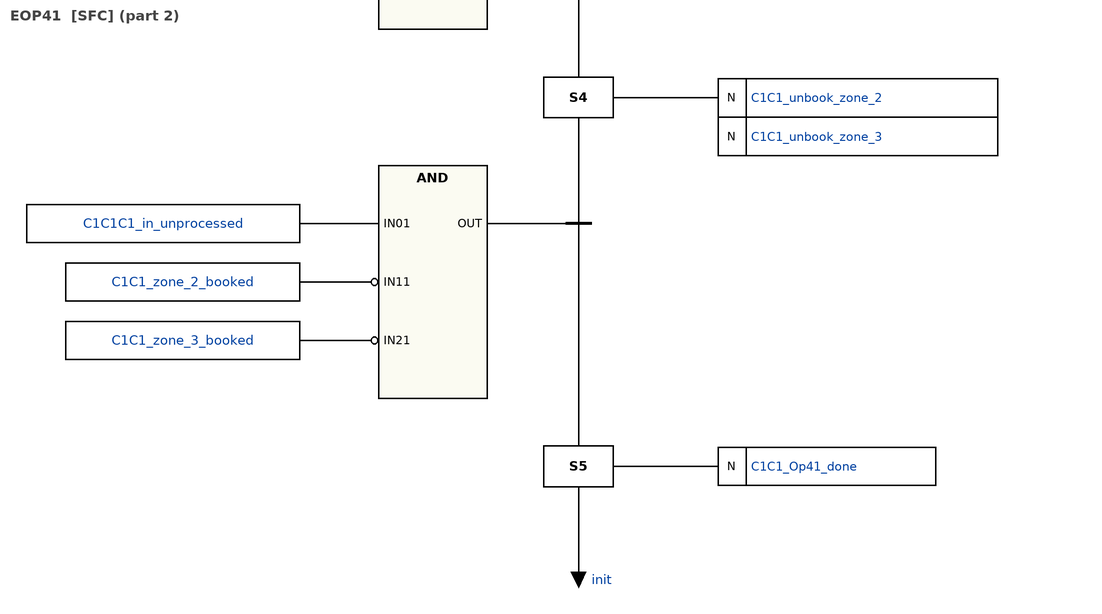
(* [picture p24: EOP41, SFC] *)
INITIAL_STEP init:
  COMPUTE_FUNCTION_BLOCKS(S);
END_STEP
TRANSITION FROM init TO S1
  := C1C1_Op41_exe_start;
END_TRANSITION
STEP S1:
END_STEP
TRANSITION FROM S1 TO S2
  := TRUE_VAR;
END_TRANSITION
STEP S2:
  C1C1_book_zone_2(N);
  C1C1_book_zone_3(N);
END_STEP
TRANSITION FROM S2 TO S3
  := _AND10_OUT;
END_TRANSITION
STEP S3:
  C1C1C1_goto_unprocessed(N);
END_STEP
TRANSITION FROM S3 TO S4
  := _AND16_OUT;
END_TRANSITION
STEP S4:
  C1C1_unbook_zone_2(N);
  C1C1_unbook_zone_3(N);
END_STEP
TRANSITION FROM S4 TO S5
  := _AND23_OUT;
END_TRANSITION
STEP S5:
  C1C1_Op41_done(N);
END_STEP
ACTION COMPUTE_FUNCTION_BLOCKS:  (* blocks drawn on the SFC sheet *)
  _AND10_OUT := C1C1_zone_2_booked AND C1C1_zone_3_booked;
  _AND16_OUT := C1C1C1_in_unprocessed AND C1C1_zone_2_booked AND C1C1_zone_3_booked;
  _AND23_OUT := C1C1C1_in_unprocessed AND NOT C1C1_zone_2_booked AND NOT C1C1_zone_3_booked;
END_ACTION
END_PROGRAM

PROGRAM EOP42
  VAR_EXTERNAL
    C1C1_Op42_exe_start : BOOL := false;
    TRUE_VAR : BOOL := true;
    C1C1C1_goto_processed : BOOL := false;
    C1C1C1_in_processed : BOOL := false;
    C1C1_Op42_done : BOOL := false;
  END_VAR

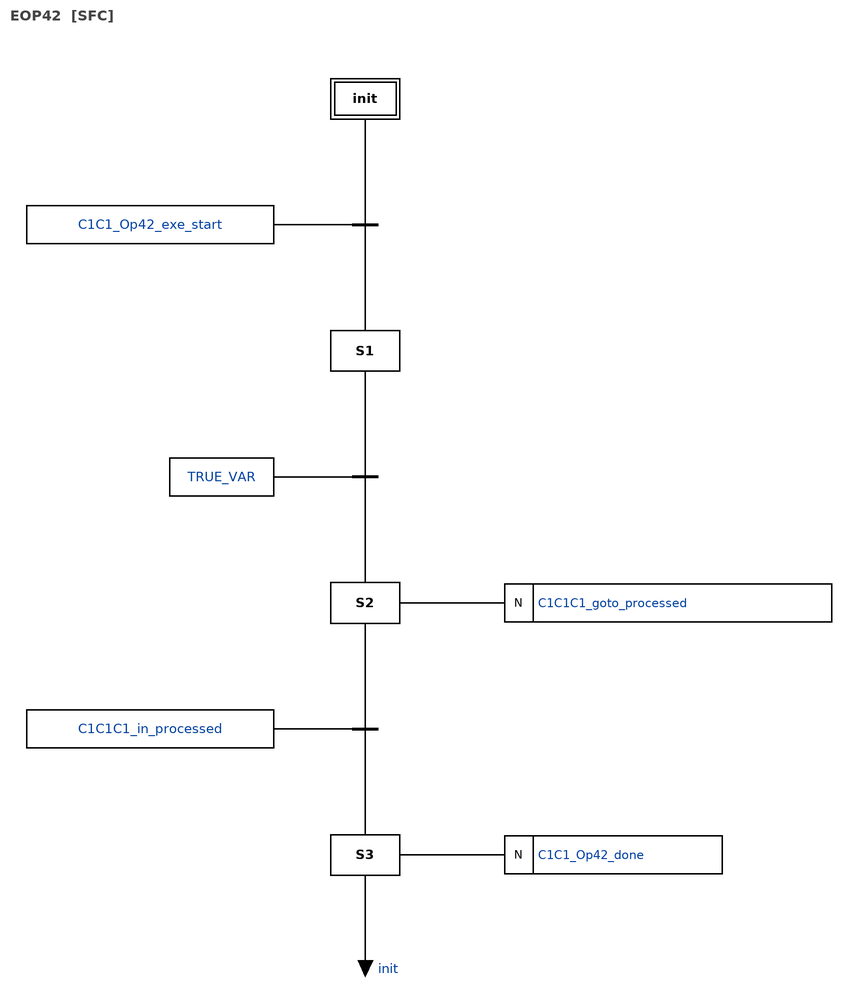
INITIAL_STEP init:
END_STEP
TRANSITION FROM init TO S1
  := C1C1_Op42_exe_start;
END_TRANSITION
STEP S1:
END_STEP
TRANSITION FROM S1 TO S2
  := TRUE_VAR;
END_TRANSITION
STEP S2:
  C1C1C1_goto_processed(N);
END_STEP
TRANSITION FROM S2 TO S3
  := C1C1C1_in_processed;
END_TRANSITION
STEP S3:
  C1C1_Op42_done(N);
END_STEP
END_PROGRAM

PROGRAM COP_C1C1_A
  VAR_EXTERNAL
    Start_COPs : BOOL := false;
    CC_A : BOOL := false;
    C1C1_Op40_exe_start : BOOL := false;
    C1C1_Op40_done : BOOL := false;
    C1C1_Op41_exe_start : BOOL := false;
    Op_34_end : BOOL := false;
    C1C1_Op41_done : BOOL := false;
    C1C1_Op42_exe_start : BOOL := false;
    C1C1_Op42_done : BOOL := false;
    COP_C1C1_A_done : BOOL := false;
    All_COP_Done_CC_A : BOOL := false;
  END_VAR
  VAR  (* added by the conversion: wires and edge detectors of the diagram *)
    _AND3_OUT : BOOL;
    _AND13_OUT : BOOL;
  END_VAR

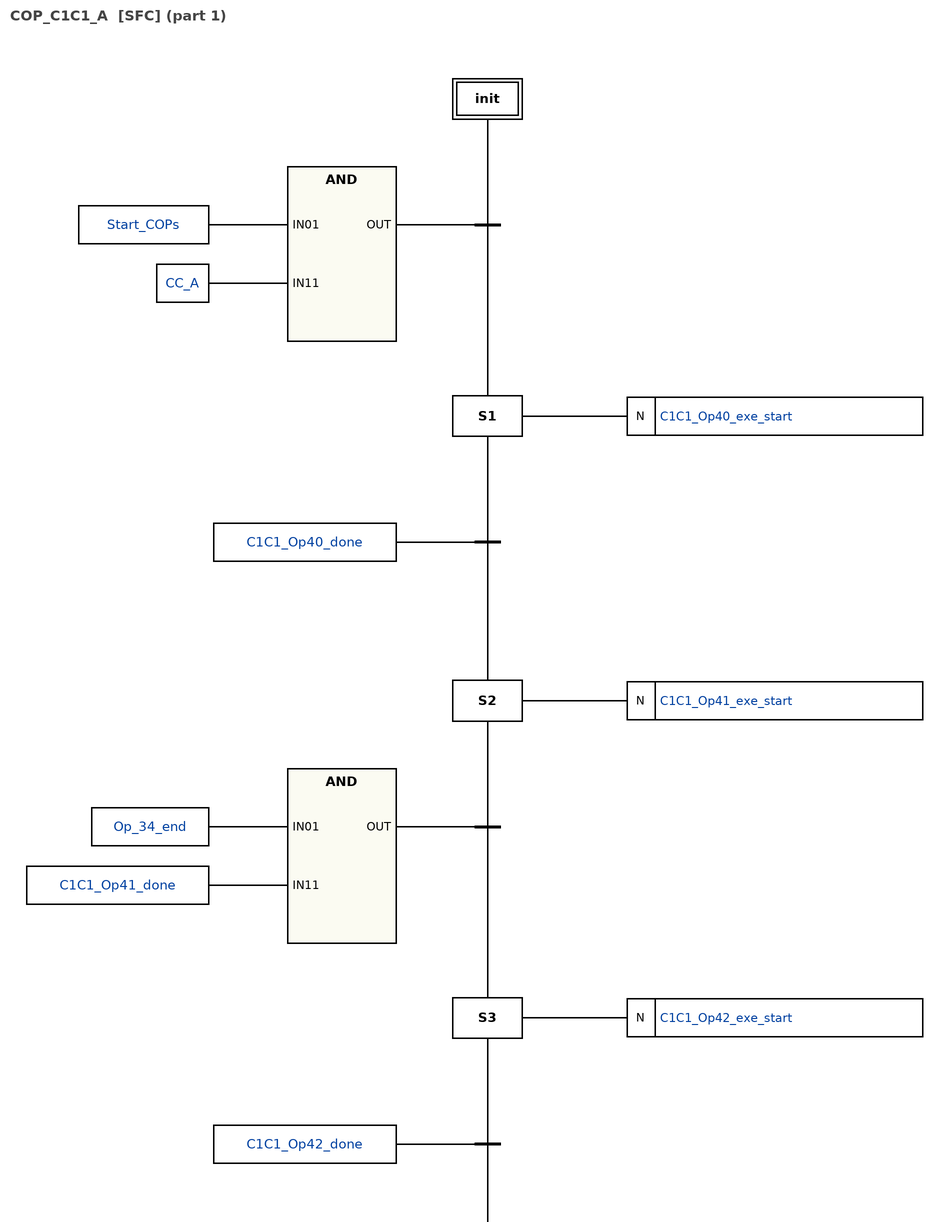
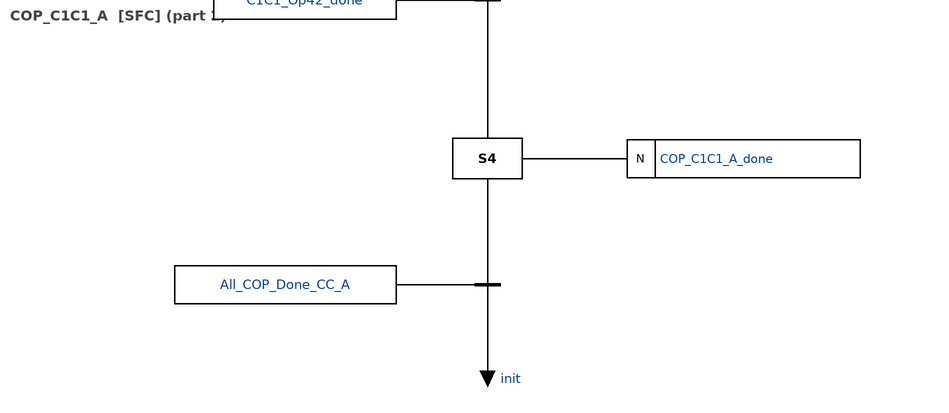
INITIAL_STEP init:
  COMPUTE_FUNCTION_BLOCKS(S);
END_STEP
TRANSITION FROM init TO S1
  := _AND3_OUT;
END_TRANSITION
STEP S1:
  C1C1_Op40_exe_start(N);
END_STEP
TRANSITION FROM S1 TO S2
  := C1C1_Op40_done;
END_TRANSITION
STEP S2:
  C1C1_Op41_exe_start(N);
END_STEP
TRANSITION FROM S2 TO S3
  := _AND13_OUT;
END_TRANSITION
STEP S3:
  C1C1_Op42_exe_start(N);
END_STEP
TRANSITION FROM S3 TO S4
  := C1C1_Op42_done;
END_TRANSITION
STEP S4:
  COP_C1C1_A_done(N);
END_STEP
TRANSITION FROM S4 TO init
  := All_COP_Done_CC_A;
END_TRANSITION
ACTION COMPUTE_FUNCTION_BLOCKS:  (* blocks drawn on the SFC sheet *)
  _AND3_OUT := Start_COPs AND CC_A;
  _AND13_OUT := Op_34_end AND C1C1_Op41_done;
END_ACTION
END_PROGRAM

PROGRAM COP_C1C1_B
  VAR_EXTERNAL
    Start_COPs : BOOL := false;
    CC_B : BOOL := false;
    C1C1_Op40_exe_start : BOOL := false;
    C1C1_Op40_done : BOOL := false;
    C1C1_Op43_exe_start : BOOL := false;
    C1C1_Op43_done : BOOL := false;
    COP_C1C1_B_done : BOOL := false;
    All_COP_Done_CC_B : BOOL := false;
  END_VAR
  VAR  (* added by the conversion: wires and edge detectors of the diagram *)
    _AND3_OUT : BOOL;
  END_VAR

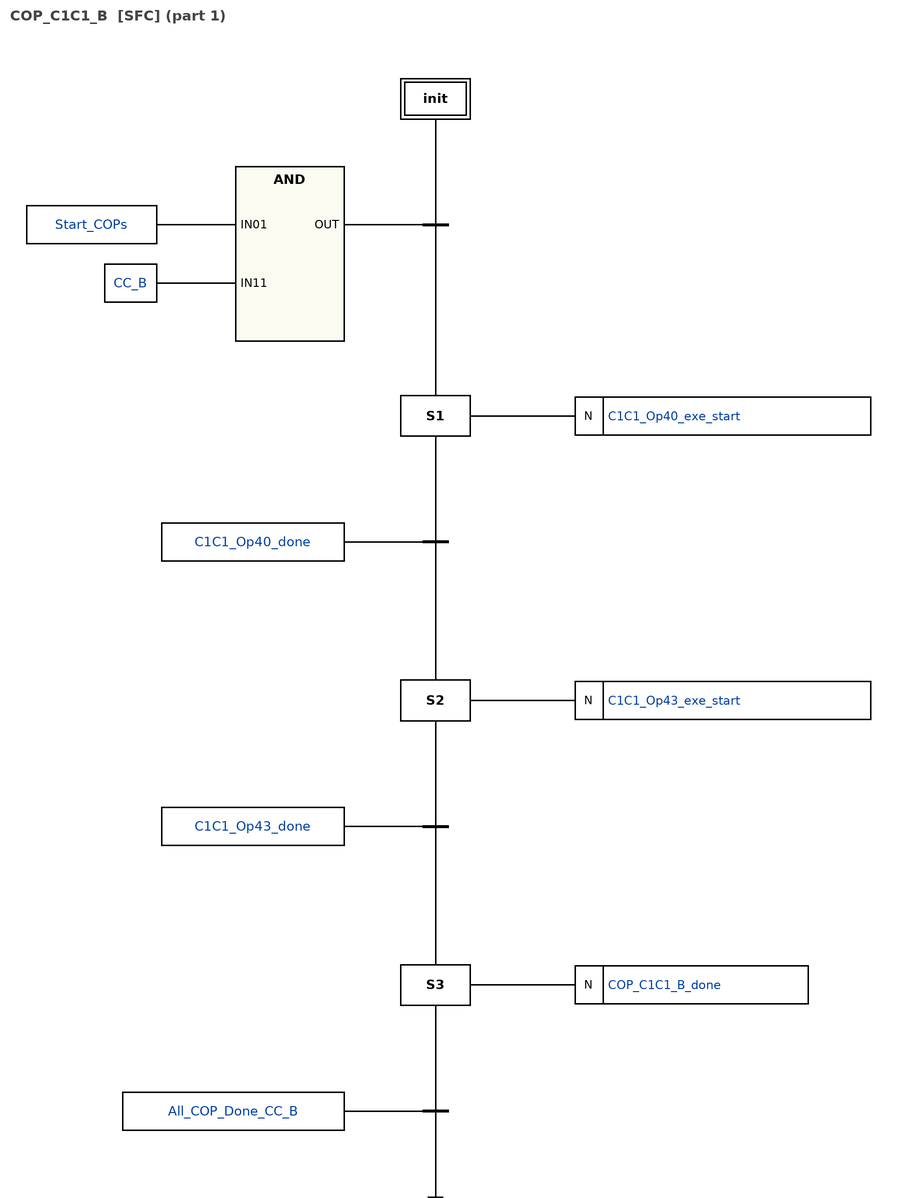
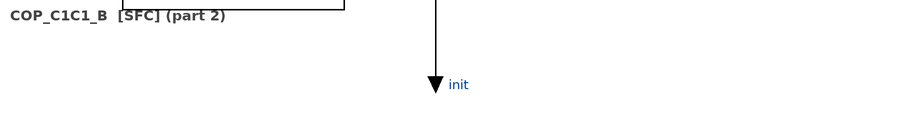
INITIAL_STEP init:
  COMPUTE_FUNCTION_BLOCKS(S);
END_STEP
TRANSITION FROM init TO S1
  := _AND3_OUT;
END_TRANSITION
STEP S1:
  C1C1_Op40_exe_start(N);
END_STEP
TRANSITION FROM S1 TO S2
  := C1C1_Op40_done;
END_TRANSITION
STEP S2:
  C1C1_Op43_exe_start(N);
END_STEP
TRANSITION FROM S2 TO S3
  := C1C1_Op43_done;
END_TRANSITION
STEP S3:
  COP_C1C1_B_done(N);
END_STEP
TRANSITION FROM S3 TO init
  := All_COP_Done_CC_B;
END_TRANSITION
ACTION COMPUTE_FUNCTION_BLOCKS:  (* blocks drawn on the SFC sheet *)
  _AND3_OUT := Start_COPs AND CC_B;
END_ACTION
END_PROGRAM

PROGRAM COP_C1C2_A
  VAR_EXTERNAL
    Start_COPs : BOOL := false;
    CC_A : BOOL := false;
    Op_10_start : BOOL := false;
    Op_10_end : BOOL := false;
    Op_11_start : BOOL := false;
    C1R1_Op21_done : BOOL := false;
    Op_11_end : BOOL := false;
    Op_12_start : BOOL := false;
    Op_12_end : BOOL := false;
    COP_C1C2_A_done : BOOL := false;
    All_COP_Done_CC_A : BOOL := false;
  END_VAR
  VAR  (* added by the conversion: wires and edge detectors of the diagram *)
    _AND3_OUT : BOOL;
    _AND13_OUT : BOOL;
  END_VAR

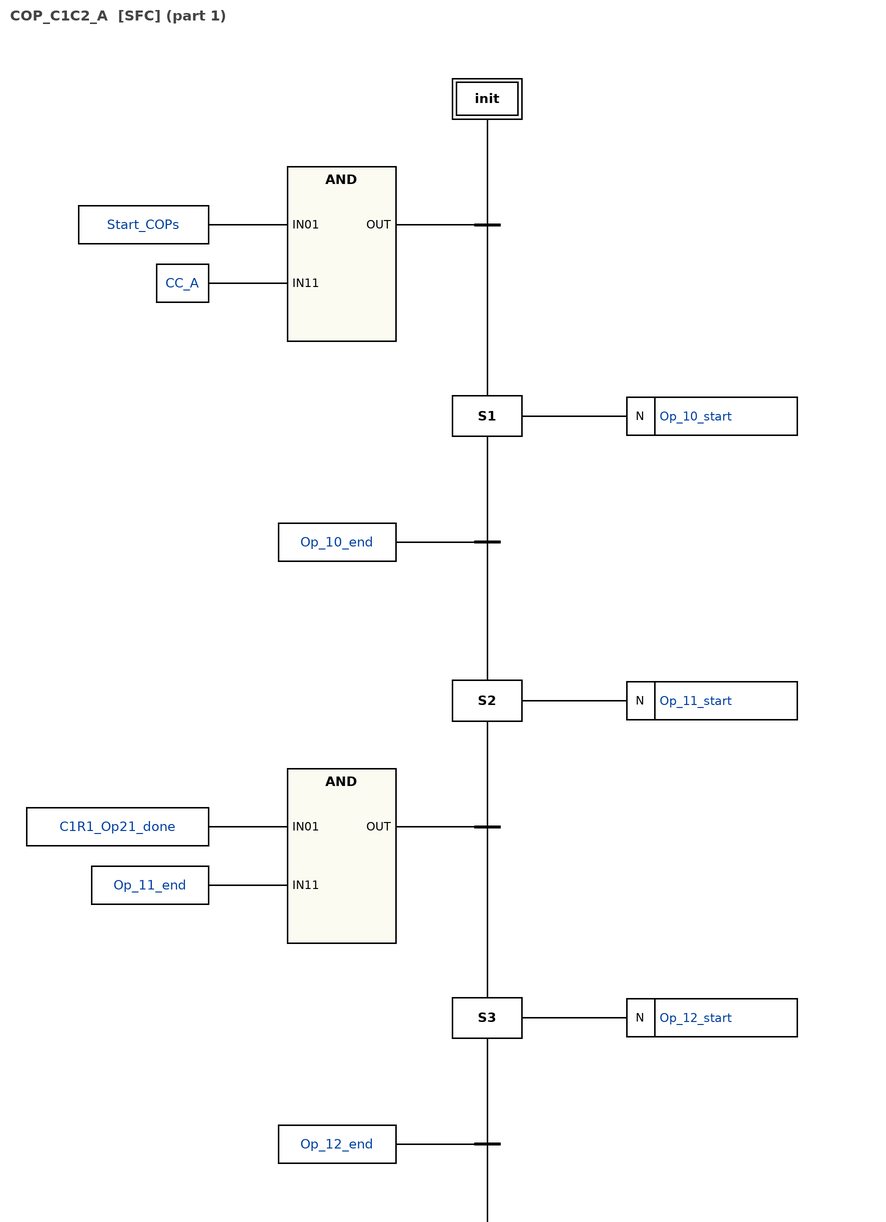
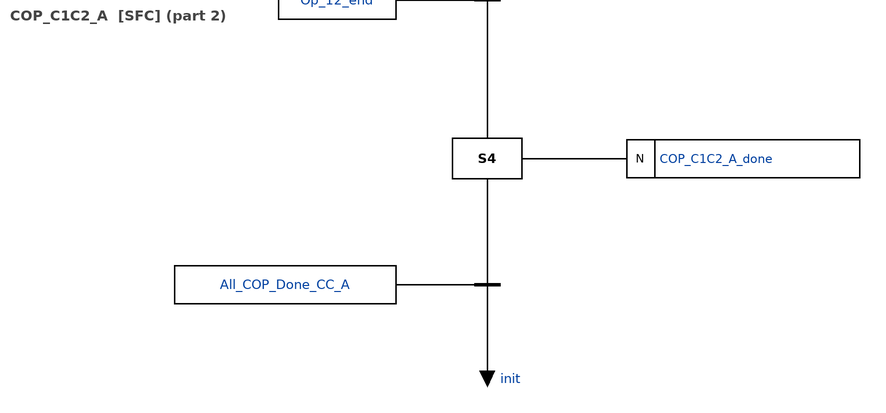
INITIAL_STEP init:
  COMPUTE_FUNCTION_BLOCKS(S);
END_STEP
TRANSITION FROM init TO S1
  := _AND3_OUT;
END_TRANSITION
STEP S1:
  Op_10_start(N);
END_STEP
TRANSITION FROM S1 TO S2
  := Op_10_end;
END_TRANSITION
STEP S2:
  Op_11_start(N);
END_STEP
TRANSITION FROM S2 TO S3
  := _AND13_OUT;
END_TRANSITION
STEP S3:
  Op_12_start(N);
END_STEP
TRANSITION FROM S3 TO S4
  := Op_12_end;
END_TRANSITION
STEP S4:
  COP_C1C2_A_done(N);
END_STEP
TRANSITION FROM S4 TO init
  := All_COP_Done_CC_A;
END_TRANSITION
ACTION COMPUTE_FUNCTION_BLOCKS:  (* blocks drawn on the SFC sheet *)
  _AND3_OUT := Start_COPs AND CC_A;
  _AND13_OUT := C1R1_Op21_done AND Op_11_end;
END_ACTION
END_PROGRAM

PROGRAM COP_C1C2_B
  VAR_EXTERNAL
    Start_COPs : BOOL := false;
    CC_B : BOOL := false;
    Op_10_start : BOOL := false;
    Op_10_end : BOOL := false;
    COP_C1C2_B_done : BOOL := false;
    All_COP_Done_CC_B : BOOL := false;
  END_VAR
  VAR  (* added by the conversion: wires and edge detectors of the diagram *)
    _AND3_OUT : BOOL;
  END_VAR

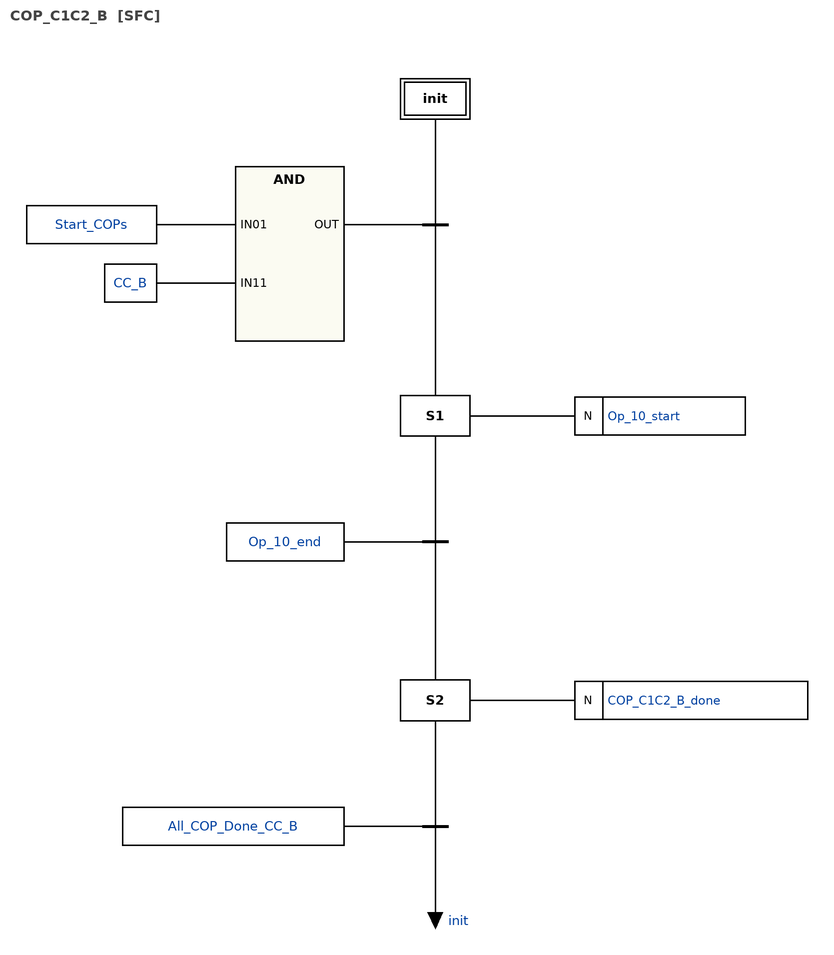
INITIAL_STEP init:
  COMPUTE_FUNCTION_BLOCKS(S);
END_STEP
TRANSITION FROM init TO S1
  := _AND3_OUT;
END_TRANSITION
STEP S1:
  Op_10_start(N);
END_STEP
TRANSITION FROM S1 TO S2
  := Op_10_end;
END_TRANSITION
STEP S2:
  COP_C1C2_B_done(N);
END_STEP
TRANSITION FROM S2 TO init
  := All_COP_Done_CC_B;
END_TRANSITION
ACTION COMPUTE_FUNCTION_BLOCKS:  (* blocks drawn on the SFC sheet *)
  _AND3_OUT := Start_COPs AND CC_B;
END_ACTION
END_PROGRAM

PROGRAM COP_C1F1_A
  VAR_EXTERNAL
    Start_COPs : BOOL := false;
    CC_A : BOOL := false;
    Op_30_start : BOOL := false;
    Op_30_end : BOOL := false;
    Op_31_start : BOOL := false;
    C1R1_Op22_done : BOOL := false;
    Op_31_end : BOOL := false;
    Op_32_start : BOOL := false;
    C1R1_Op23_done : BOOL := false;
    Op_32_end : BOOL := false;
    Op_33_start : BOOL := false;
    C1R1_Op24_done : BOOL := false;
    Op_33_end : BOOL := false;
    COP_C1F1_A_done : BOOL := false;
    All_COP_Done_CC_A : BOOL := false;
  END_VAR
  VAR  (* added by the conversion: wires and edge detectors of the diagram *)
    _AND3_OUT : BOOL;
    _AND13_OUT : BOOL;
    _AND19_OUT : BOOL;
    _AND25_OUT : BOOL;
  END_VAR

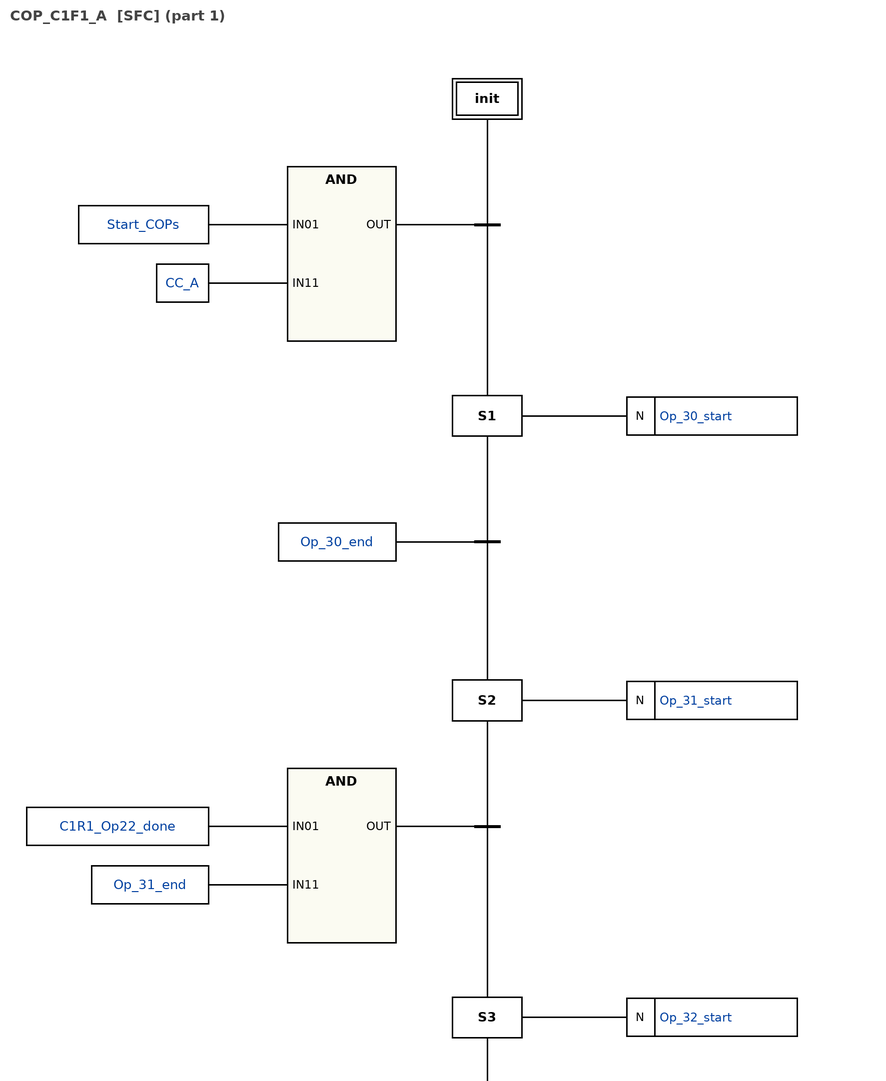
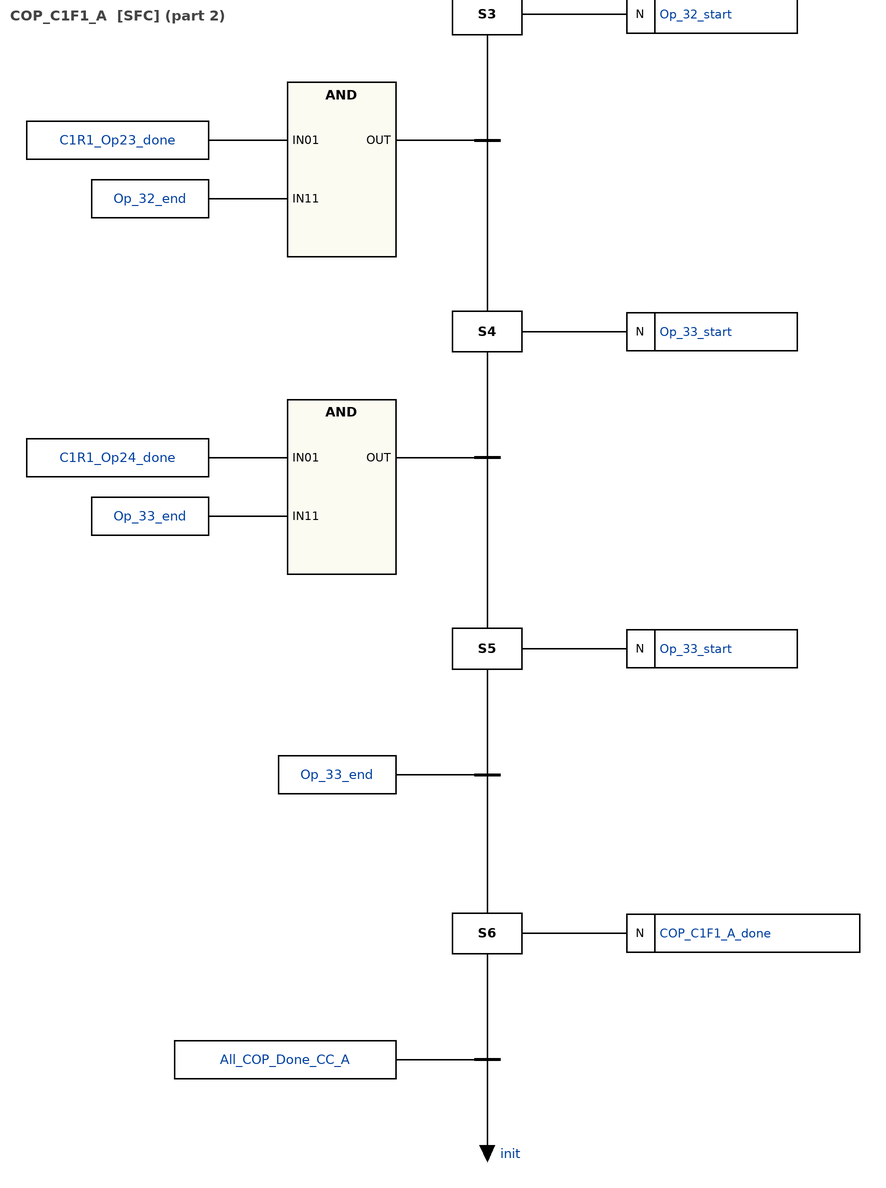
INITIAL_STEP init:
  COMPUTE_FUNCTION_BLOCKS(S);
END_STEP
TRANSITION FROM init TO S1
  := _AND3_OUT;
END_TRANSITION
STEP S1:
  Op_30_start(N);
END_STEP
TRANSITION FROM S1 TO S2
  := Op_30_end;
END_TRANSITION
STEP S2:
  Op_31_start(N);
END_STEP
TRANSITION FROM S2 TO S3
  := _AND13_OUT;
END_TRANSITION
STEP S3:
  Op_32_start(N);
END_STEP
TRANSITION FROM S3 TO S4
  := _AND19_OUT;
END_TRANSITION
STEP S4:
  Op_33_start(N);
END_STEP
TRANSITION FROM S4 TO S5
  := _AND25_OUT;
END_TRANSITION
STEP S5:
  Op_33_start(N);
END_STEP
TRANSITION FROM S5 TO S6
  := Op_33_end;
END_TRANSITION
STEP S6:
  COP_C1F1_A_done(N);
END_STEP
TRANSITION FROM S6 TO init
  := All_COP_Done_CC_A;
END_TRANSITION
ACTION COMPUTE_FUNCTION_BLOCKS:  (* blocks drawn on the SFC sheet *)
  _AND3_OUT := Start_COPs AND CC_A;
  _AND13_OUT := C1R1_Op22_done AND Op_31_end;
  _AND19_OUT := C1R1_Op23_done AND Op_32_end;
  _AND25_OUT := C1R1_Op24_done AND Op_33_end;
END_ACTION
END_PROGRAM

PROGRAM COP_C1F1_B
  VAR_EXTERNAL
    Start_COPs : BOOL := false;
    CC_B : BOOL := false;
    Op_30_start : BOOL := false;
    Op_30_end : BOOL := false;
    COP_C1F1_B_done : BOOL := false;
    All_COP_Done_CC_B : BOOL := false;
  END_VAR
  VAR  (* added by the conversion: wires and edge detectors of the diagram *)
    _AND3_OUT : BOOL;
  END_VAR

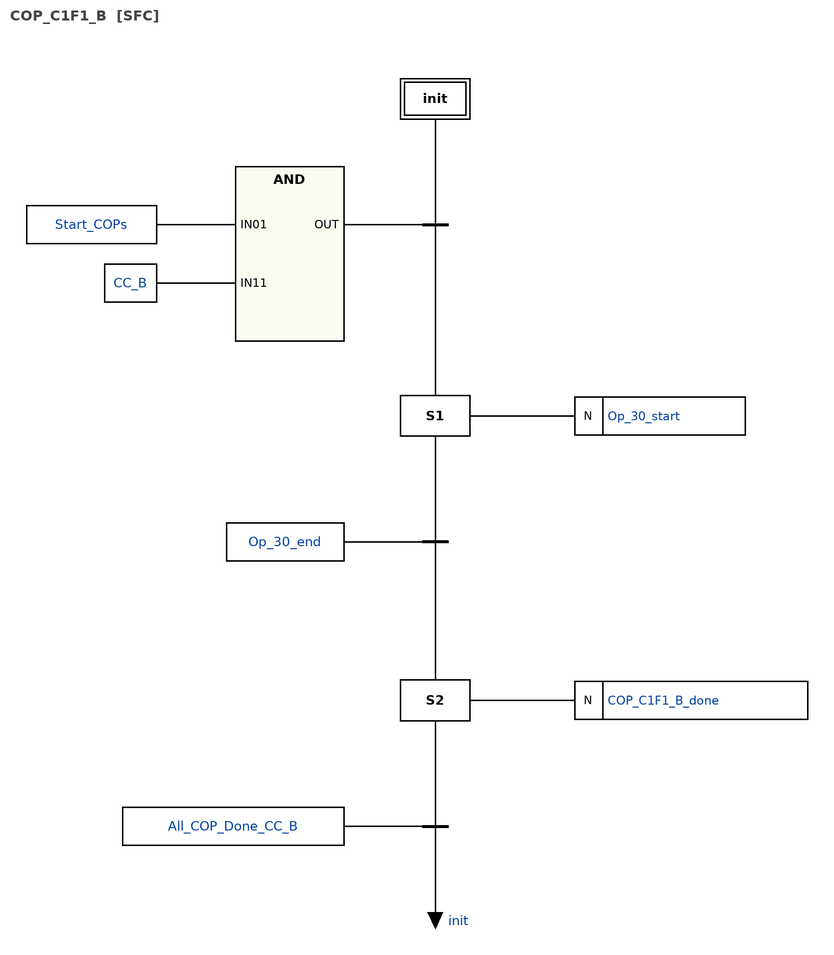
INITIAL_STEP init:
  COMPUTE_FUNCTION_BLOCKS(S);
END_STEP
TRANSITION FROM init TO S1
  := _AND3_OUT;
END_TRANSITION
STEP S1:
  Op_30_start(N);
END_STEP
TRANSITION FROM S1 TO S2
  := Op_30_end;
END_TRANSITION
STEP S2:
  COP_C1F1_B_done(N);
END_STEP
TRANSITION FROM S2 TO init
  := All_COP_Done_CC_B;
END_TRANSITION
ACTION COMPUTE_FUNCTION_BLOCKS:  (* blocks drawn on the SFC sheet *)
  _AND3_OUT := Start_COPs AND CC_B;
END_ACTION
END_PROGRAM

PROGRAM COP_C1R1_A
  VAR_EXTERNAL
    Start_COPs : BOOL := false;
    CC_A : BOOL := false;
    C1R1_Op20_exe_start : BOOL := false;
    Op_11_end : BOOL := false;
    C1R1_Op20_done : BOOL := false;
    C1R1_Op21_exe_start : BOOL := false;
    Op_31_end : BOOL := false;
    C1R1_Op21_done : BOOL := false;
    C1R1_Op22_exe_start : BOOL := false;
    Op_32_end : BOOL := false;
    C1R1_Op22_done : BOOL := false;
    C1R1_Op23_exe_start : BOOL := false;
    Op_33_end : BOOL := false;
    C1R1_Op23_done : BOOL := false;
    C1R1_Op24_exe_start : BOOL := false;
    C1R1_Op24_done : BOOL := false;
    COP_C1R1_A_done : BOOL := false;
    All_COP_Done_CC_A : BOOL := false;
  END_VAR
  VAR  (* added by the conversion: wires and edge detectors of the diagram *)
    _AND3_OUT : BOOL;
    _AND9_OUT : BOOL;
    _AND15_OUT : BOOL;
    _AND21_OUT : BOOL;
    _AND27_OUT : BOOL;
  END_VAR

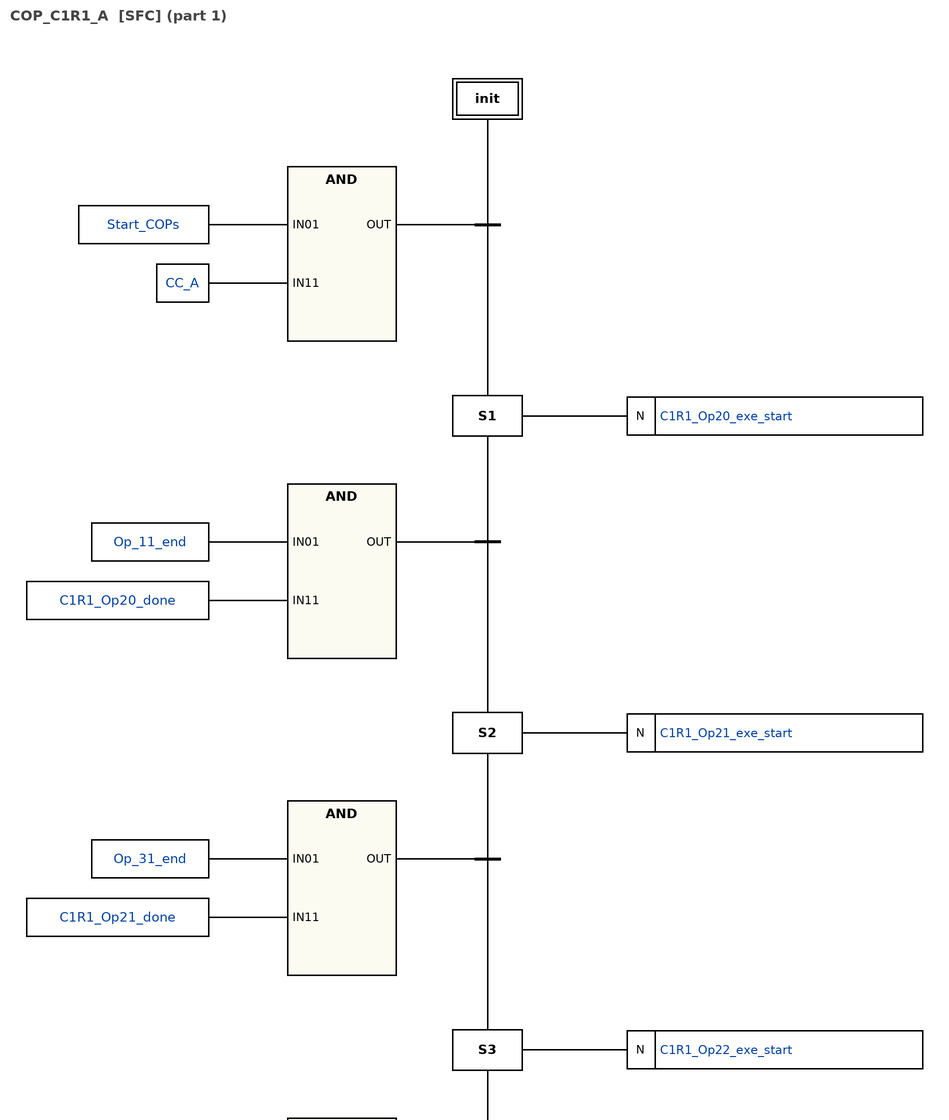
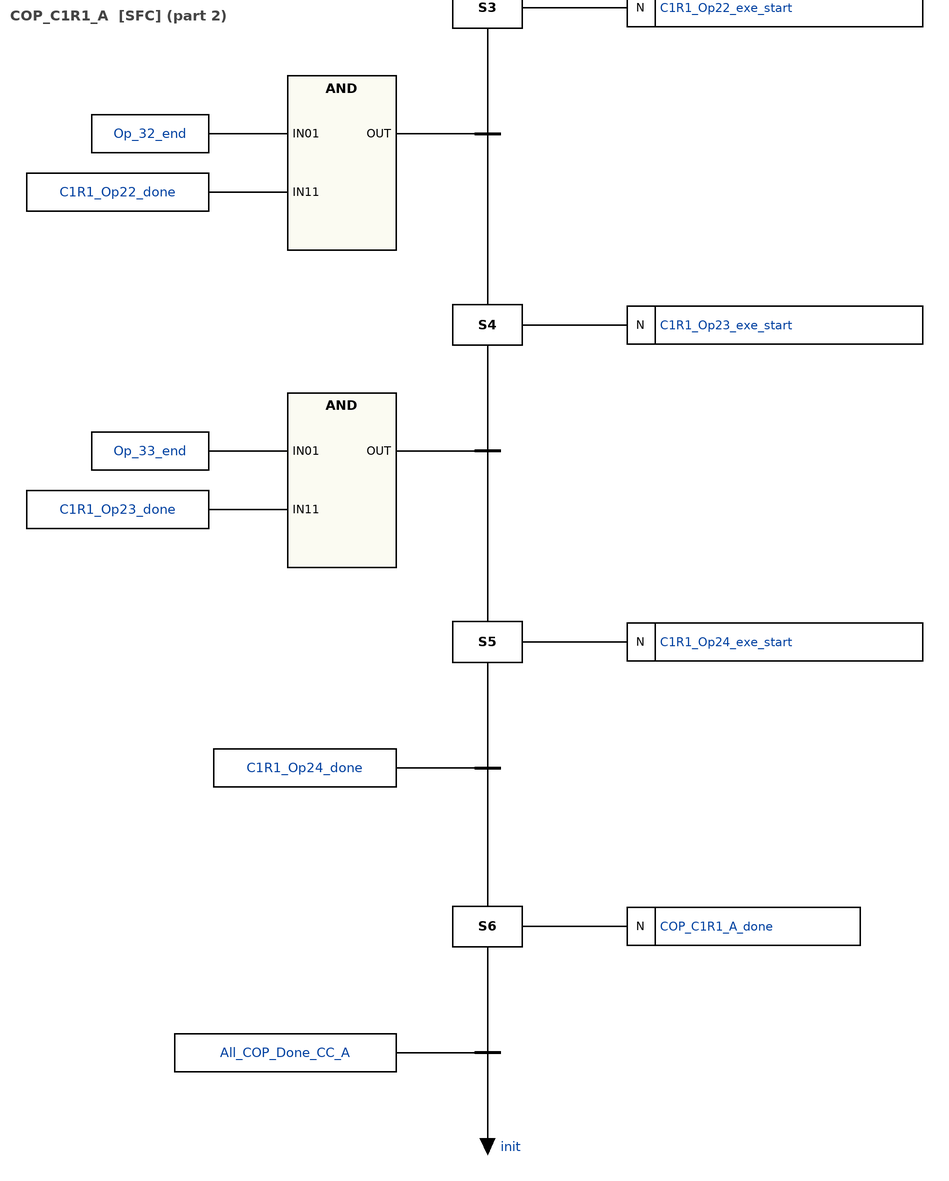
INITIAL_STEP init:
  COMPUTE_FUNCTION_BLOCKS(S);
END_STEP
TRANSITION FROM init TO S1
  := _AND3_OUT;
END_TRANSITION
STEP S1:
  C1R1_Op20_exe_start(N);
END_STEP
TRANSITION FROM S1 TO S2
  := _AND9_OUT;
END_TRANSITION
STEP S2:
  C1R1_Op21_exe_start(N);
END_STEP
TRANSITION FROM S2 TO S3
  := _AND15_OUT;
END_TRANSITION
STEP S3:
  C1R1_Op22_exe_start(N);
END_STEP
TRANSITION FROM S3 TO S4
  := _AND21_OUT;
END_TRANSITION
STEP S4:
  C1R1_Op23_exe_start(N);
END_STEP
TRANSITION FROM S4 TO S5
  := _AND27_OUT;
END_TRANSITION
STEP S5:
  C1R1_Op24_exe_start(N);
END_STEP
TRANSITION FROM S5 TO S6
  := C1R1_Op24_done;
END_TRANSITION
STEP S6:
  COP_C1R1_A_done(N);
END_STEP
TRANSITION FROM S6 TO init
  := All_COP_Done_CC_A;
END_TRANSITION
ACTION COMPUTE_FUNCTION_BLOCKS:  (* blocks drawn on the SFC sheet *)
  _AND3_OUT := Start_COPs AND CC_A;
  _AND9_OUT := Op_11_end AND C1R1_Op20_done;
  _AND15_OUT := Op_31_end AND C1R1_Op21_done;
  _AND21_OUT := Op_32_end AND C1R1_Op22_done;
  _AND27_OUT := Op_33_end AND C1R1_Op23_done;
END_ACTION
END_PROGRAM

PROGRAM FB_C1R1_External_Machine_comm_-_5_OP
  VAR_EXTERNAL
    C1R1_Op20_exe : BOOL := false;
    C1R1_Op20_IL : BOOL := false;
    C1R1_Op20_done : BOOL := false;
    C1R1_Op20_started : BOOL := false;
    C1R1_Op21_exe : BOOL := false;
    C1R1_Op21_IL : BOOL := false;
    C1R1_Op21_done : BOOL := false;
    C1R1_Op21_started : BOOL := false;
    C1R1_Op22_exe : BOOL := false;
    C1R1_Op22_IL : BOOL := false;
    C1R1_Op22_done : BOOL := false;
    C1R1_Op22_started : BOOL := false;
    C1R1_Op23_exe : BOOL := false;
    C1R1_Op23_IL : BOOL := false;
    C1R1_Op23_done : BOOL := false;
    C1R1_Op23_started : BOOL := false;
    C1R1_Op24_exe : BOOL := false;
    C1R1_Op24_IL : BOOL := false;
    C1R1_Op24_done : BOOL := false;
    C1R1_Op24_started : BOOL := false;
    C1R1_ext_lb_0 : BOOL := false;
    C1R1_ext_Ob_0 : BOOL := false;
    C1R1_ext_lb_1 : BOOL := false;
    C1R1_ext_Ob_1 : BOOL := false;
    C1R1_ext_lb_2 : BOOL := false;
    C1R1_ext_Ob_2 : BOOL := false;
    C1R1_ext_lb_3 : BOOL := false;
    C1R1_ext_Ob_3 : BOOL := false;
    C1R1_ext_lb_4 : BOOL := false;
    C1R1_ext_Ob_4 : BOOL := false;
    C1R1_ext_lb_5 : BOOL := false;
    C1R1_ext_Ob_5 : BOOL := false;
    C1R1_ext_lb_6 : BOOL := false;
    C1R1_ext_Ob_6 : BOOL := false;
    C1R1_ext_lb_7 : BOOL := false;
    C1R1_ext_Ob_7 : BOOL := false;
    C1R1_ext_machine_OK : BOOL := false;
    C1R1_IL_OK : BOOL := false;
  END_VAR
  VAR_EXTERNAL CONSTANT
    Constant_20 : INT := 20;
    Constant_21 : INT := 21;
    Constant_22 : INT := 22;
    Constant_23 : INT := 23;
    Constant_24 : INT := 24;
  END_VAR
  VAR
    FB_C1R1_External_Machine_comm_-_5_OP : External Machine comm - 5 OP;
  END_VAR

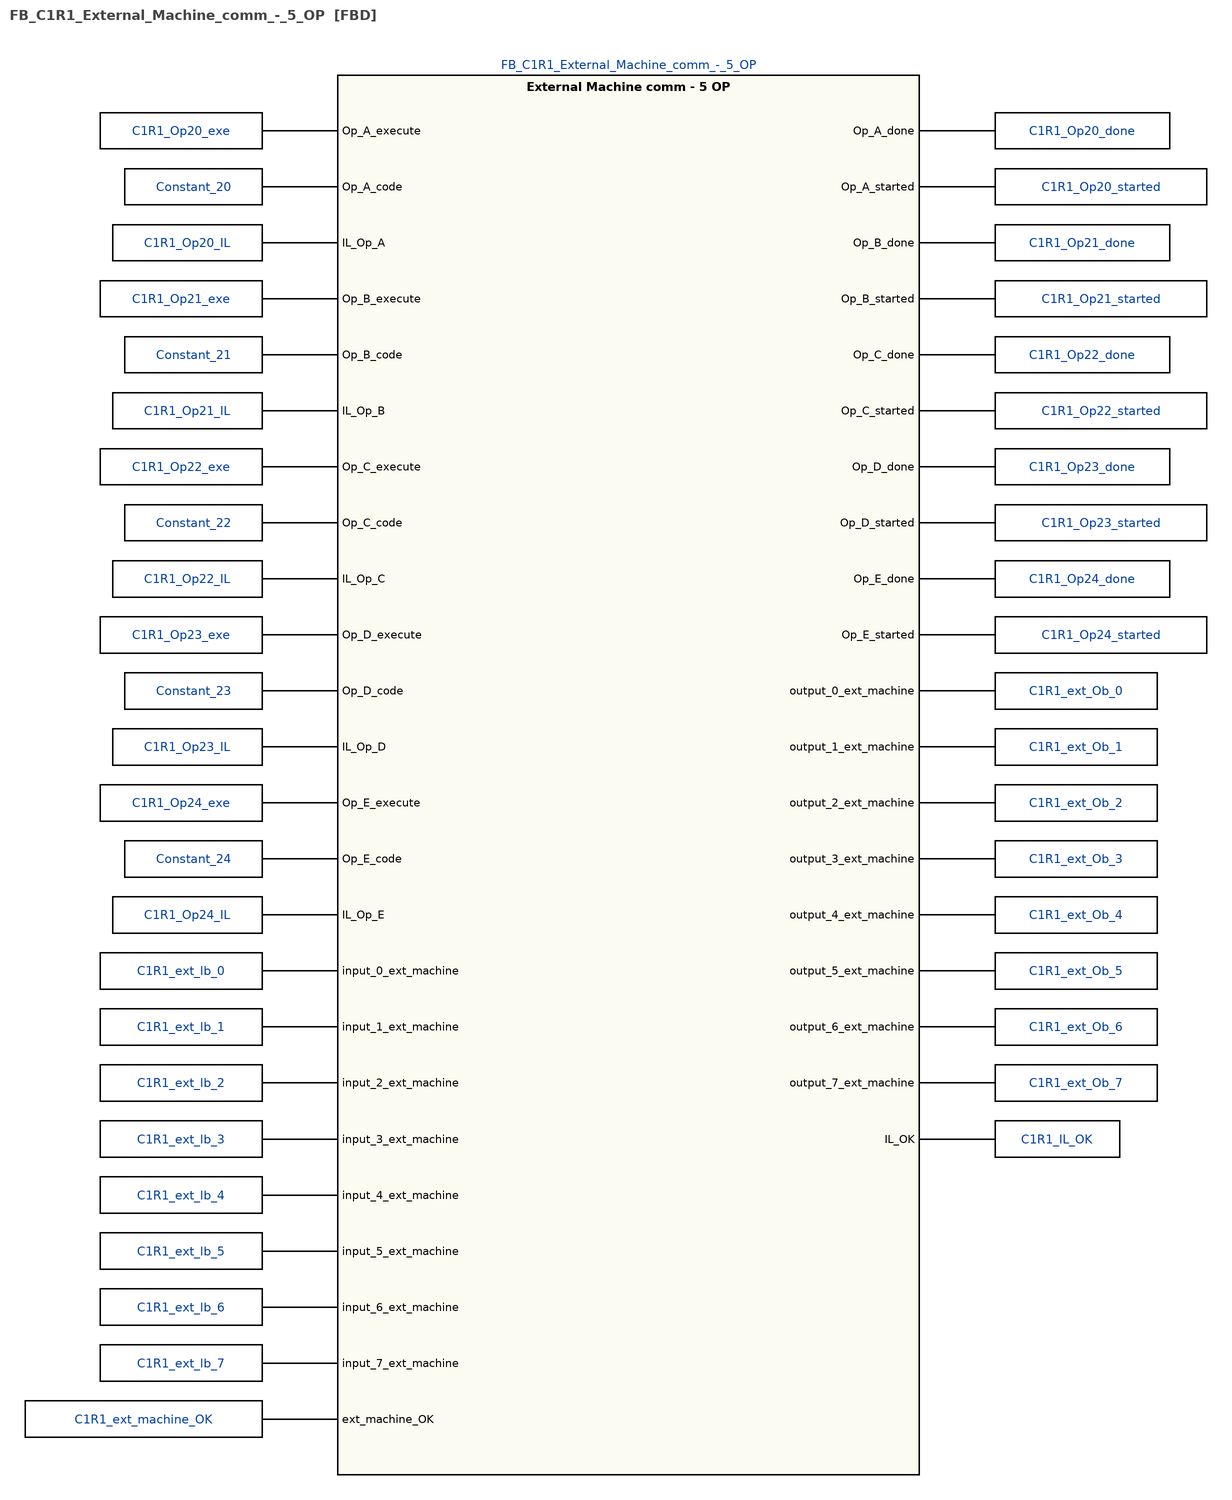
(* FBD diagram, written out as Structured Text *)
FB_C1R1_External_Machine_comm_-_5_OP(Op_A_execute := C1R1_Op20_exe, Op_A_code := Constant_20, IL_Op_A := C1R1_Op20_IL, Op_B_execute := C1R1_Op21_exe, Op_B_code := Constant_21, IL_Op_B := C1R1_Op21_IL, Op_C_execute := C1R1_Op22_exe, Op_C_code := Constant_22, IL_Op_C := C1R1_Op22_IL, Op_D_execute := C1R1_Op23_exe, Op_D_code := Constant_23, IL_Op_D := C1R1_Op23_IL, Op_E_execute := C1R1_Op24_exe, Op_E_code := Constant_24, IL_Op_E := C1R1_Op24_IL, input_0_ext_machine := C1R1_ext_lb_0, input_1_ext_machine := C1R1_ext_lb_1, input_2_ext_machine := C1R1_ext_lb_2, input_3_ext_machine := C1R1_ext_lb_3, input_4_ext_machine := C1R1_ext_lb_4, input_5_ext_machine := C1R1_ext_lb_5, input_6_ext_machine := C1R1_ext_lb_6, input_7_ext_machine := C1R1_ext_lb_7, ext_machine_OK := C1R1_ext_machine_OK);
C1R1_Op20_done := FB_C1R1_External_Machine_comm_-_5_OP.Op_A_done;
C1R1_Op20_started := FB_C1R1_External_Machine_comm_-_5_OP.Op_A_started;
C1R1_Op21_done := FB_C1R1_External_Machine_comm_-_5_OP.Op_B_done;
C1R1_Op21_started := FB_C1R1_External_Machine_comm_-_5_OP.Op_B_started;
C1R1_Op22_done := FB_C1R1_External_Machine_comm_-_5_OP.Op_C_done;
C1R1_Op22_started := FB_C1R1_External_Machine_comm_-_5_OP.Op_C_started;
C1R1_Op23_done := FB_C1R1_External_Machine_comm_-_5_OP.Op_D_done;
C1R1_Op23_started := FB_C1R1_External_Machine_comm_-_5_OP.Op_D_started;
C1R1_Op24_done := FB_C1R1_External_Machine_comm_-_5_OP.Op_E_done;
C1R1_Op24_started := FB_C1R1_External_Machine_comm_-_5_OP.Op_E_started;
C1R1_ext_Ob_0 := FB_C1R1_External_Machine_comm_-_5_OP.output_0_ext_machine;
C1R1_ext_Ob_1 := FB_C1R1_External_Machine_comm_-_5_OP.output_1_ext_machine;
C1R1_ext_Ob_2 := FB_C1R1_External_Machine_comm_-_5_OP.output_2_ext_machine;
C1R1_ext_Ob_3 := FB_C1R1_External_Machine_comm_-_5_OP.output_3_ext_machine;
C1R1_ext_Ob_4 := FB_C1R1_External_Machine_comm_-_5_OP.output_4_ext_machine;
C1R1_ext_Ob_5 := FB_C1R1_External_Machine_comm_-_5_OP.output_5_ext_machine;
C1R1_ext_Ob_6 := FB_C1R1_External_Machine_comm_-_5_OP.output_6_ext_machine;
C1R1_ext_Ob_7 := FB_C1R1_External_Machine_comm_-_5_OP.output_7_ext_machine;
C1R1_IL_OK := FB_C1R1_External_Machine_comm_-_5_OP.IL_OK;
END_PROGRAM

PROGRAM FB_C1C1_External_Machine_comm_-_4_OP
  VAR_EXTERNAL
    C1C1_Op40_exe : BOOL := false;
    C1C1_Op40_IL : BOOL := false;
    C1C1_Op40_done : BOOL := false;
    C1C1_Op40_started : BOOL := false;
    C1C1_Op41_exe : BOOL := false;
    C1C1_Op41_IL : BOOL := false;
    C1C1_Op41_done : BOOL := false;
    C1C1_Op41_started : BOOL := false;
    C1C1_Op42_exe : BOOL := false;
    C1C1_Op42_IL : BOOL := false;
    C1C1_Op42_done : BOOL := false;
    C1C1_Op42_started : BOOL := false;
    C1C1_Op43_exe : BOOL := false;
    C1C1_Op43_IL : BOOL := false;
    C1C1_Op43_done : BOOL := false;
    C1C1_Op43_started : BOOL := false;
    C1C1_ext_lb_0 : BOOL := false;
    C1C1_ext_Ob_0 : BOOL := false;
    C1C1_ext_lb_1 : BOOL := false;
    C1C1_ext_Ob_1 : BOOL := false;
    C1C1_ext_lb_2 : BOOL := false;
    C1C1_ext_Ob_2 : BOOL := false;
    C1C1_ext_lb_3 : BOOL := false;
    C1C1_ext_Ob_3 : BOOL := false;
    C1C1_ext_lb_4 : BOOL := false;
    C1C1_ext_Ob_4 : BOOL := false;
    C1C1_ext_lb_5 : BOOL := false;
    C1C1_ext_Ob_5 : BOOL := false;
    C1C1_ext_lb_6 : BOOL := false;
    C1C1_ext_Ob_6 : BOOL := false;
    C1C1_ext_lb_7 : BOOL := false;
    C1C1_ext_Ob_7 : BOOL := false;
    C1C1_ext_machine_OK : BOOL := false;
    C1C1_IL_OK : BOOL := false;
  END_VAR
  VAR_EXTERNAL CONSTANT
    Constant_40 : INT := 40;
    Constant_41 : INT := 41;
    Constant_42 : INT := 42;
    Constant_43 : INT := 43;
  END_VAR
  VAR
    FB_C1C1_External_Machine_comm_-_4_OP : External Machine comm - 4 OP;
  END_VAR

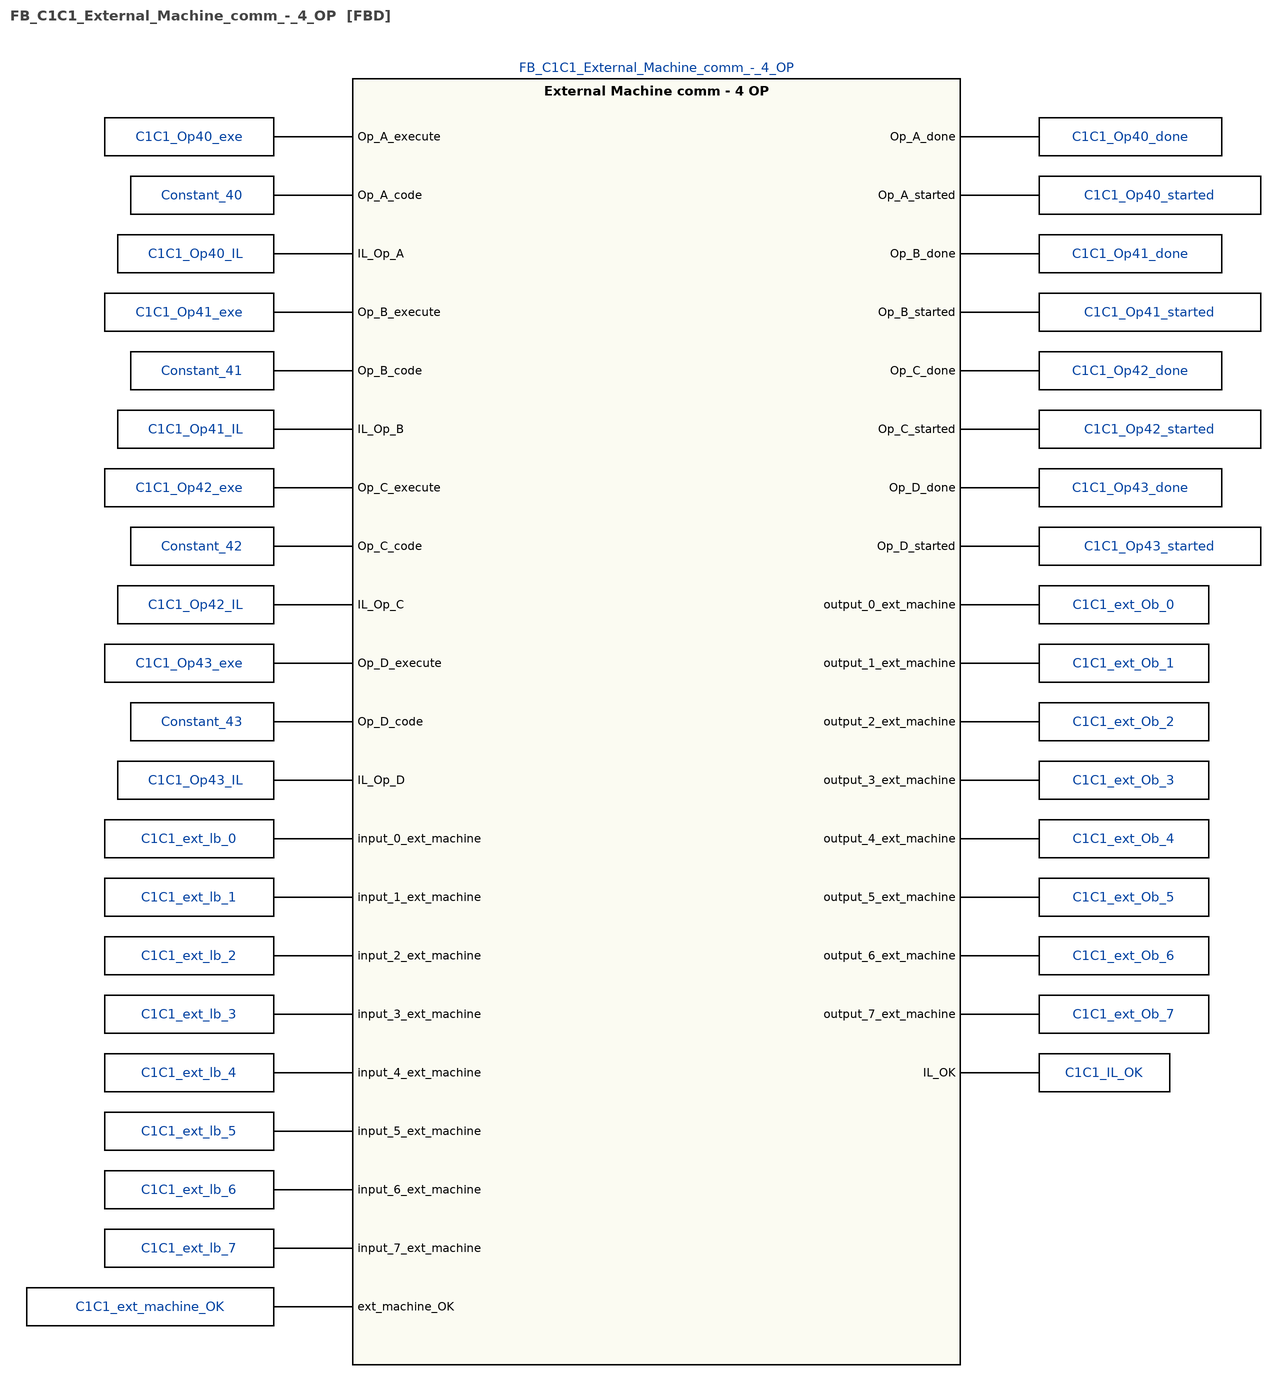
(* FBD diagram, written out as Structured Text *)
FB_C1C1_External_Machine_comm_-_4_OP(Op_A_execute := C1C1_Op40_exe, Op_A_code := Constant_40, IL_Op_A := C1C1_Op40_IL, Op_B_execute := C1C1_Op41_exe, Op_B_code := Constant_41, IL_Op_B := C1C1_Op41_IL, Op_C_execute := C1C1_Op42_exe, Op_C_code := Constant_42, IL_Op_C := C1C1_Op42_IL, Op_D_execute := C1C1_Op43_exe, Op_D_code := Constant_43, IL_Op_D := C1C1_Op43_IL, input_0_ext_machine := C1C1_ext_lb_0, input_1_ext_machine := C1C1_ext_lb_1, input_2_ext_machine := C1C1_ext_lb_2, input_3_ext_machine := C1C1_ext_lb_3, input_4_ext_machine := C1C1_ext_lb_4, input_5_ext_machine := C1C1_ext_lb_5, input_6_ext_machine := C1C1_ext_lb_6, input_7_ext_machine := C1C1_ext_lb_7, ext_machine_OK := C1C1_ext_machine_OK);
C1C1_Op40_done := FB_C1C1_External_Machine_comm_-_4_OP.Op_A_done;
C1C1_Op40_started := FB_C1C1_External_Machine_comm_-_4_OP.Op_A_started;
C1C1_Op41_done := FB_C1C1_External_Machine_comm_-_4_OP.Op_B_done;
C1C1_Op41_started := FB_C1C1_External_Machine_comm_-_4_OP.Op_B_started;
C1C1_Op42_done := FB_C1C1_External_Machine_comm_-_4_OP.Op_C_done;
C1C1_Op42_started := FB_C1C1_External_Machine_comm_-_4_OP.Op_C_started;
C1C1_Op43_done := FB_C1C1_External_Machine_comm_-_4_OP.Op_D_done;
C1C1_Op43_started := FB_C1C1_External_Machine_comm_-_4_OP.Op_D_started;
C1C1_ext_Ob_0 := FB_C1C1_External_Machine_comm_-_4_OP.output_0_ext_machine;
C1C1_ext_Ob_1 := FB_C1C1_External_Machine_comm_-_4_OP.output_1_ext_machine;
C1C1_ext_Ob_2 := FB_C1C1_External_Machine_comm_-_4_OP.output_2_ext_machine;
C1C1_ext_Ob_3 := FB_C1C1_External_Machine_comm_-_4_OP.output_3_ext_machine;
C1C1_ext_Ob_4 := FB_C1C1_External_Machine_comm_-_4_OP.output_4_ext_machine;
C1C1_ext_Ob_5 := FB_C1C1_External_Machine_comm_-_4_OP.output_5_ext_machine;
C1C1_ext_Ob_6 := FB_C1C1_External_Machine_comm_-_4_OP.output_6_ext_machine;
C1C1_ext_Ob_7 := FB_C1C1_External_Machine_comm_-_4_OP.output_7_ext_machine;
C1C1_IL_OK := FB_C1C1_External_Machine_comm_-_4_OP.IL_OK;
END_PROGRAM

PROGRAM FB_C1C2C1_Belt_Conveyor
  VAR_EXTERNAL
    C1C2C1_in_part_in_position : BOOL := false;
    C1C2C1_goto_part_in_position : BOOL := false;
    C1C2C1_IL_to_part_in_position : BOOL := false;
    C1C2C1_to_part_in_position_started : BOOL := false;
    C1C2C1_QS1 : BOOL := false;
    C1C2C1_in_position_empty : BOOL := false;
    C1C2C1_goto_position_empty : BOOL := false;
    C1C2C1_IL_to_position_empty : BOOL := false;
    C1C2C1_to_position_empty_started : BOOL := false;
    C1C2C1_QS2 : BOOL := false;
    Not_Connected : BOOL := false;
  END_VAR
  VAR
    FB_C1C2C1_Belt_Conveyor : Belt Conveyor;
  END_VAR

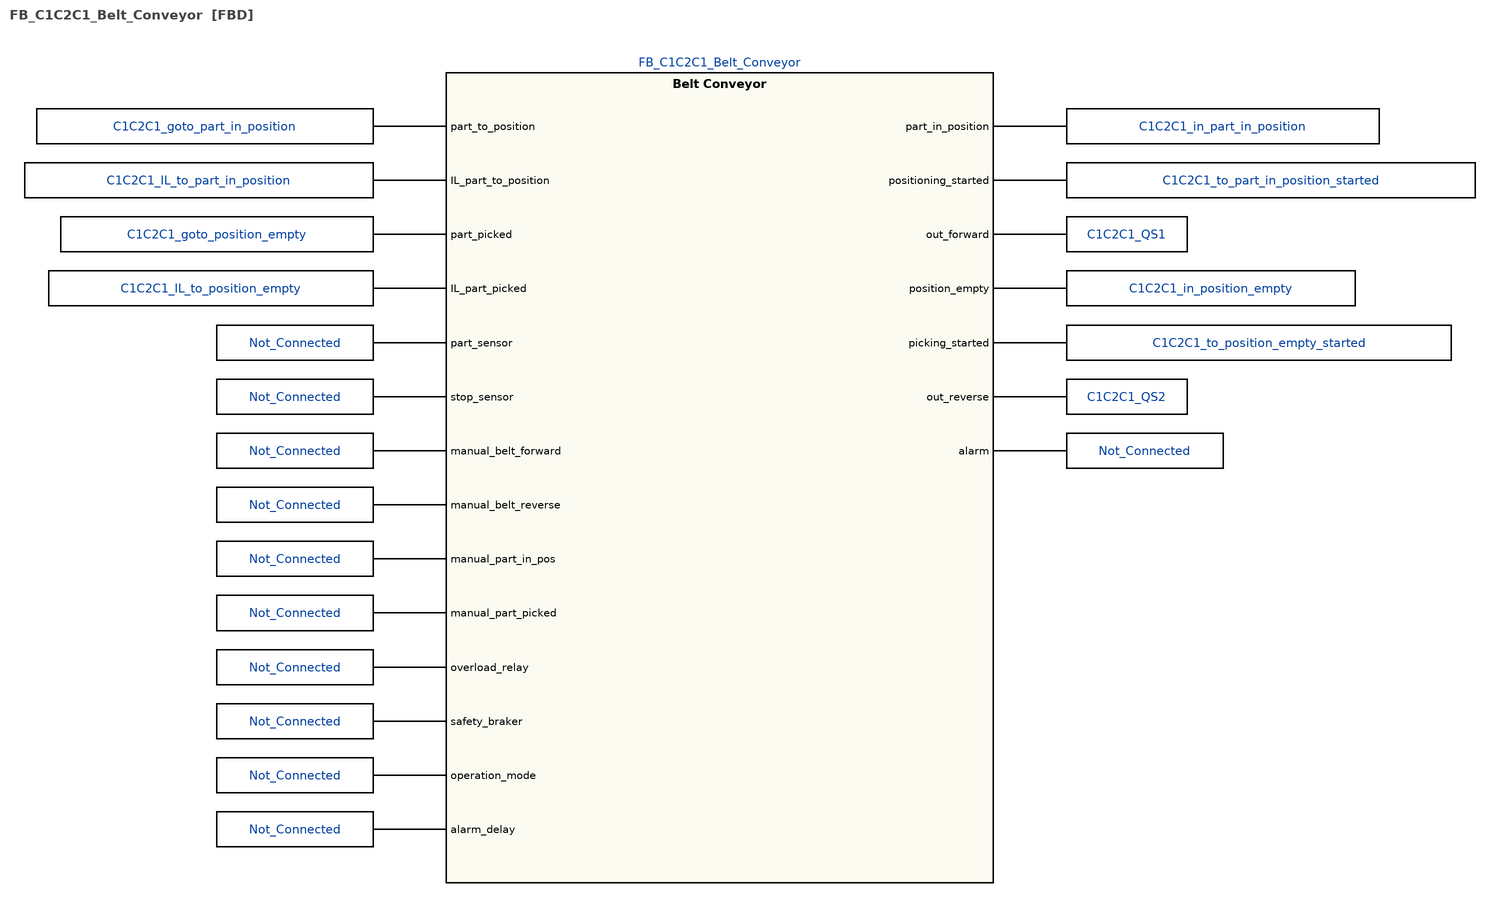
(* FBD diagram, written out as Structured Text *)
FB_C1C2C1_Belt_Conveyor(part_to_position := C1C2C1_goto_part_in_position, IL_part_to_position := C1C2C1_IL_to_part_in_position, part_picked := C1C2C1_goto_position_empty, IL_part_picked := C1C2C1_IL_to_position_empty, part_sensor := Not_Connected, stop_sensor := Not_Connected, manual_belt_forward := Not_Connected, manual_belt_reverse := Not_Connected, manual_part_in_pos := Not_Connected, manual_part_picked := Not_Connected, overload_relay := Not_Connected, safety_braker := Not_Connected, operation_mode := Not_Connected, alarm_delay := Not_Connected);
C1C2C1_in_part_in_position := FB_C1C2C1_Belt_Conveyor.part_in_position;
C1C2C1_to_part_in_position_started := FB_C1C2C1_Belt_Conveyor.positioning_started;
C1C2C1_QS1 := FB_C1C2C1_Belt_Conveyor.out_forward;
C1C2C1_in_position_empty := FB_C1C2C1_Belt_Conveyor.position_empty;
C1C2C1_to_position_empty_started := FB_C1C2C1_Belt_Conveyor.picking_started;
C1C2C1_QS2 := FB_C1C2C1_Belt_Conveyor.out_reverse;
Not_Connected := FB_C1C2C1_Belt_Conveyor.alarm;
END_PROGRAM

PROGRAM FB_C1F1C1_Two_Position_Movement
  VAR_EXTERNAL
    C1F1C1_in_home : BOOL := false;
    C1F1C1_goto_home : BOOL := false;
    C1F1C1_IL_to_home : BOOL := false;
    C1F1C1_to_home_started : BOOL := false;
    C1F1C1_QS1 : BOOL := false;
    C1F1C1_IS1 : BOOL := false;
    C1F1C1_in_work_pos : BOOL := false;
    C1F1C1_goto_work_pos : BOOL := false;
    C1F1C1_IL_to_work_pos : BOOL := false;
    C1F1C1_to_work_pos_started : BOOL := false;
    C1F1C1_QS2 : BOOL := false;
    C1F1C1_IS2 : BOOL := false;
    Not_Connected : BOOL := false;
  END_VAR
  VAR
    FB_C1F1C1_Two_Position_Movement : Two Position Movement;
  END_VAR

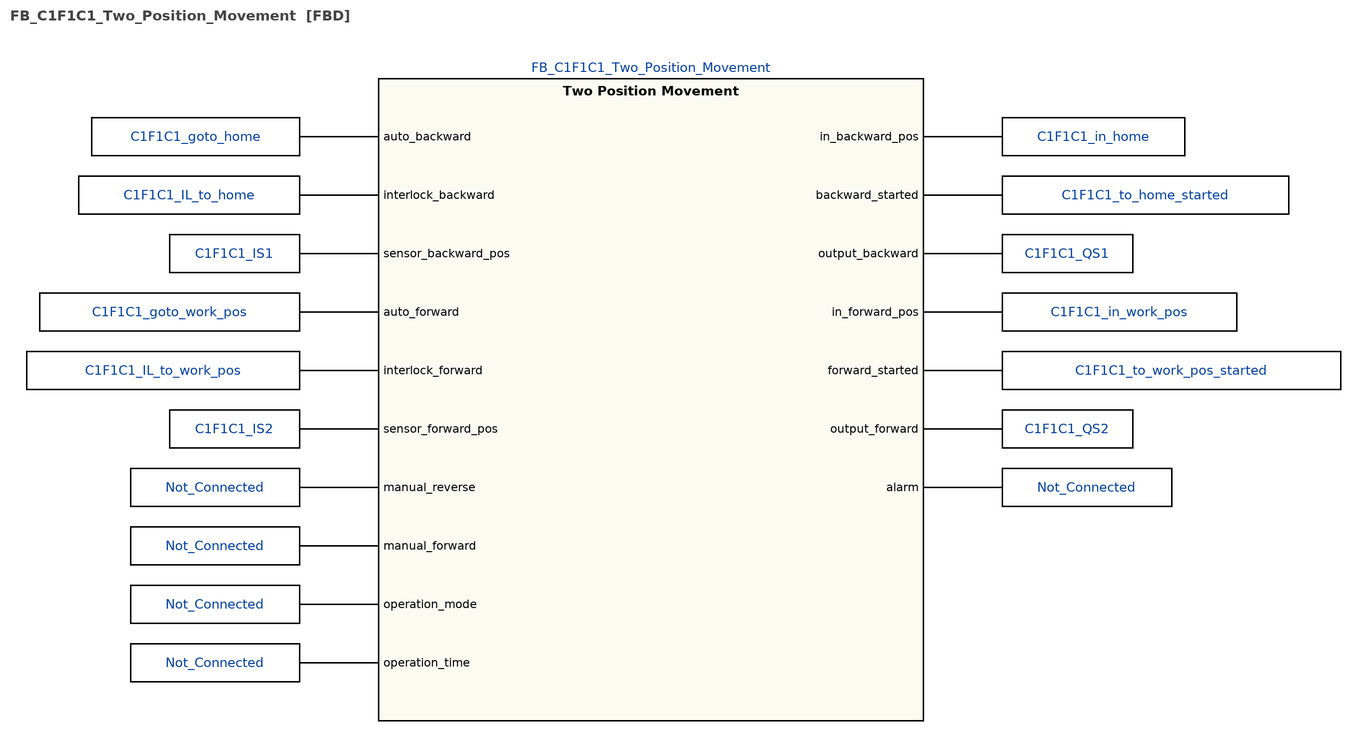
(* FBD diagram, written out as Structured Text *)
FB_C1F1C1_Two_Position_Movement(auto_backward := C1F1C1_goto_home, interlock_backward := C1F1C1_IL_to_home, sensor_backward_pos := C1F1C1_IS1, auto_forward := C1F1C1_goto_work_pos, interlock_forward := C1F1C1_IL_to_work_pos, sensor_forward_pos := C1F1C1_IS2, manual_reverse := Not_Connected, manual_forward := Not_Connected, operation_mode := Not_Connected, operation_time := Not_Connected);
C1F1C1_in_home := FB_C1F1C1_Two_Position_Movement.in_backward_pos;
C1F1C1_to_home_started := FB_C1F1C1_Two_Position_Movement.backward_started;
C1F1C1_QS1 := FB_C1F1C1_Two_Position_Movement.output_backward;
C1F1C1_in_work_pos := FB_C1F1C1_Two_Position_Movement.in_forward_pos;
C1F1C1_to_work_pos_started := FB_C1F1C1_Two_Position_Movement.forward_started;
C1F1C1_QS2 := FB_C1F1C1_Two_Position_Movement.output_forward;
Not_Connected := FB_C1F1C1_Two_Position_Movement.alarm;
END_PROGRAM

PROGRAM FB_C1F1C2_Two_Position_Movement
  VAR_EXTERNAL
    C1F1C2_in_locked : BOOL := false;
    C1F1C2_goto_locked : BOOL := false;
    C1F1C2_IL_to_locked : BOOL := false;
    C1F1C2_to_locked_started : BOOL := false;
    C1F1C2_QS1 : BOOL := false;
    C1F1C2_IS1 : BOOL := false;
    C1F1C2_in_unlocked : BOOL := false;
    C1F1C2_goto_unlocked : BOOL := false;
    C1F1C2_IL_to_unlocked : BOOL := false;
    C1F1C2_to_unlocked_started : BOOL := false;
    C1F1C2_QS2 : BOOL := false;
    C1F1C2_IS2 : BOOL := false;
    Not_Connected : BOOL := false;
  END_VAR
  VAR
    FB_C1F1C2_Two_Position_Movement : Two Position Movement;
  END_VAR

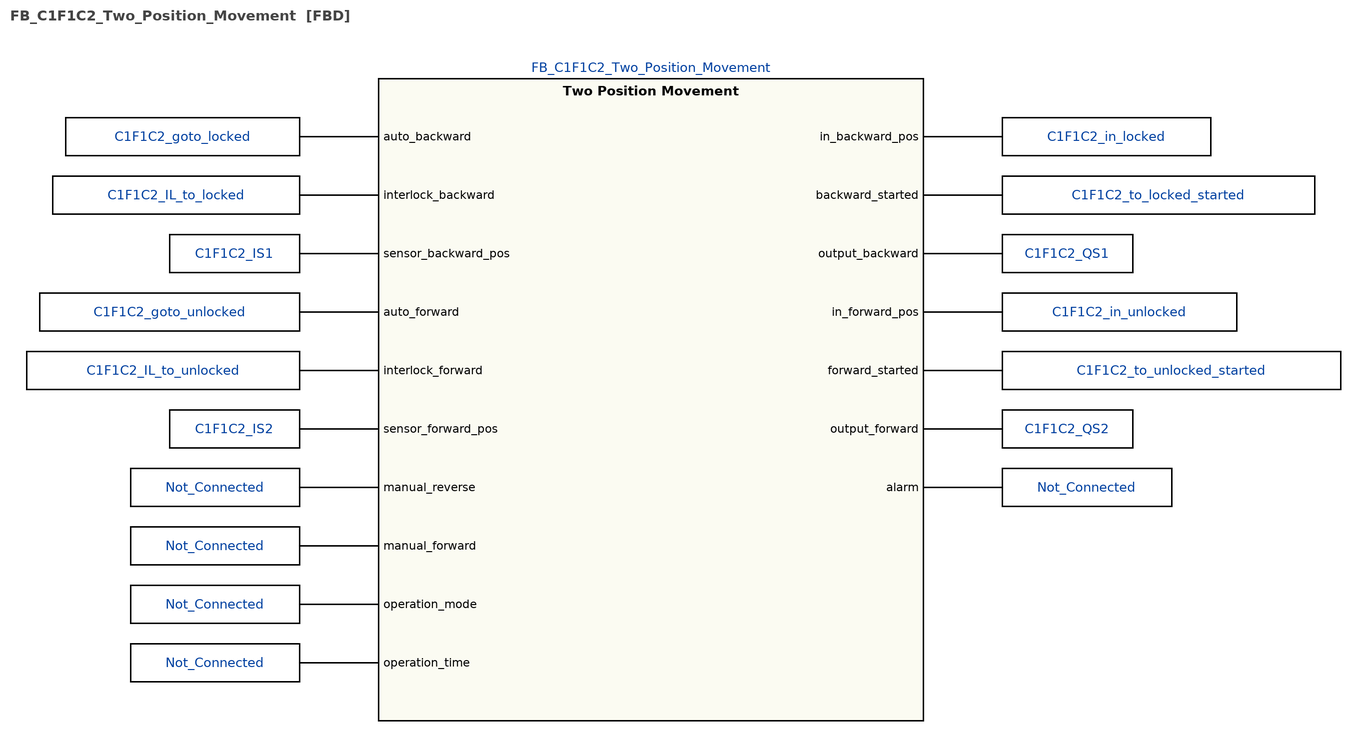
(* FBD diagram, written out as Structured Text *)
FB_C1F1C2_Two_Position_Movement(auto_backward := C1F1C2_goto_locked, interlock_backward := C1F1C2_IL_to_locked, sensor_backward_pos := C1F1C2_IS1, auto_forward := C1F1C2_goto_unlocked, interlock_forward := C1F1C2_IL_to_unlocked, sensor_forward_pos := C1F1C2_IS2, manual_reverse := Not_Connected, manual_forward := Not_Connected, operation_mode := Not_Connected, operation_time := Not_Connected);
C1F1C2_in_locked := FB_C1F1C2_Two_Position_Movement.in_backward_pos;
C1F1C2_to_locked_started := FB_C1F1C2_Two_Position_Movement.backward_started;
C1F1C2_QS1 := FB_C1F1C2_Two_Position_Movement.output_backward;
C1F1C2_in_unlocked := FB_C1F1C2_Two_Position_Movement.in_forward_pos;
C1F1C2_to_unlocked_started := FB_C1F1C2_Two_Position_Movement.forward_started;
C1F1C2_QS2 := FB_C1F1C2_Two_Position_Movement.output_forward;
Not_Connected := FB_C1F1C2_Two_Position_Movement.alarm;
END_PROGRAM

PROGRAM FB_C1F1C3_Two_Position_Movement
  VAR_EXTERNAL
    C1F1C3_in_open : BOOL := false;
    C1F1C3_goto_open : BOOL := false;
    C1F1C3_IL_to_open : BOOL := false;
    C1F1C3_to_open_started : BOOL := false;
    C1F1C3_QS1 : BOOL := false;
    C1F1C3_IS1A : BOOL := false;
    C1F1C3_IS1B : BOOL := false;
    C1F1C3_in_close : BOOL := false;
    C1F1C3_goto_close : BOOL := false;
    C1F1C3_IL_to_close : BOOL := false;
    C1F1C3_to_close_started : BOOL := false;
    C1F1C3_QS2 : BOOL := false;
    C1F1C3_IS2A : BOOL := false;
    C1F1C3_IS2B : BOOL := false;
    Not_Connected : BOOL := false;
  END_VAR
  VAR
    FB_C1F1C3_Two_Position_Movement : Two Position Movement;
  END_VAR

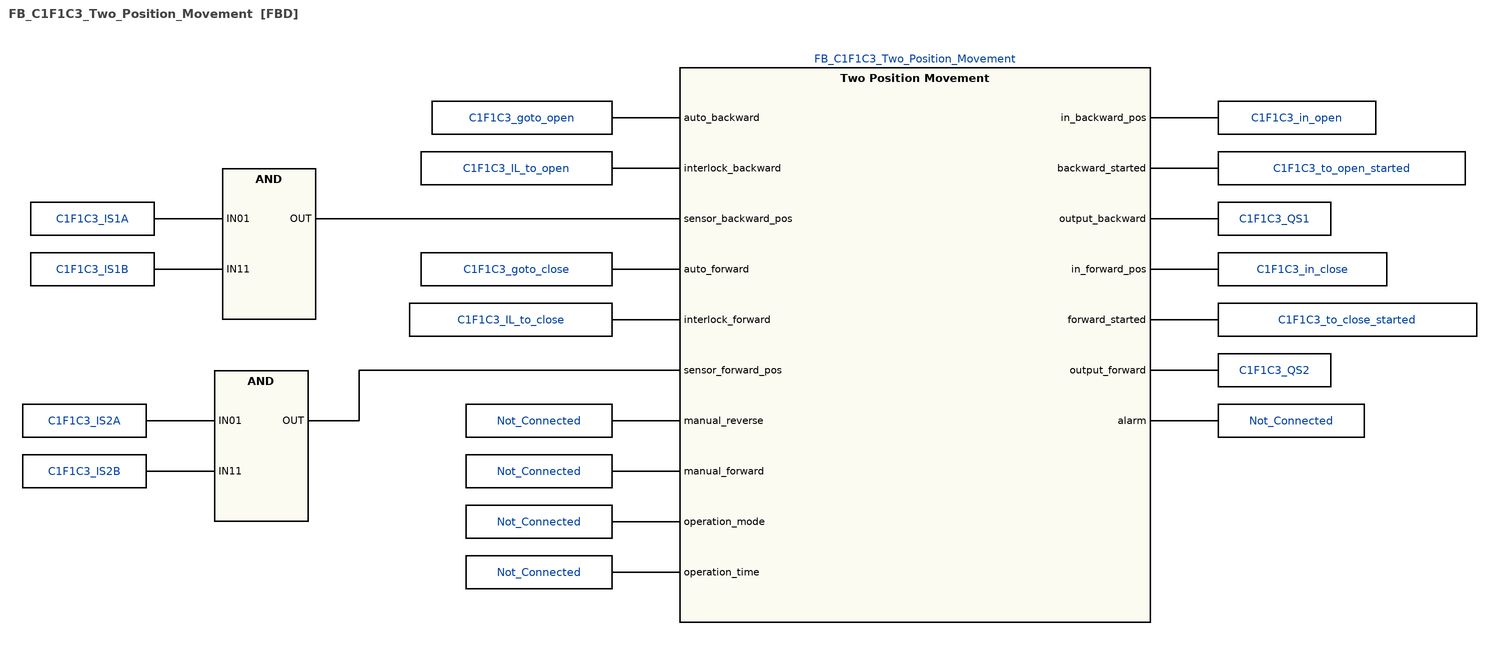
(* FBD diagram, written out as Structured Text *)
FB_C1F1C3_Two_Position_Movement(auto_backward := C1F1C3_goto_open, interlock_backward := C1F1C3_IL_to_open, sensor_backward_pos := C1F1C3_IS1A AND C1F1C3_IS1B, auto_forward := C1F1C3_goto_close, interlock_forward := C1F1C3_IL_to_close, sensor_forward_pos := C1F1C3_IS2A AND C1F1C3_IS2B, manual_reverse := Not_Connected, manual_forward := Not_Connected, operation_mode := Not_Connected, operation_time := Not_Connected);
C1F1C3_in_open := FB_C1F1C3_Two_Position_Movement.in_backward_pos;
C1F1C3_to_open_started := FB_C1F1C3_Two_Position_Movement.backward_started;
C1F1C3_QS1 := FB_C1F1C3_Two_Position_Movement.output_backward;
C1F1C3_in_close := FB_C1F1C3_Two_Position_Movement.in_forward_pos;
C1F1C3_to_close_started := FB_C1F1C3_Two_Position_Movement.forward_started;
C1F1C3_QS2 := FB_C1F1C3_Two_Position_Movement.output_forward;
Not_Connected := FB_C1F1C3_Two_Position_Movement.alarm;
END_PROGRAM

PROGRAM FB_C1F1C4_Part_Detection_x2
  VAR_EXTERNAL
    C1F1C4_in_on : BOOL := false;
    C1F1C4_in_off : BOOL := false;
    C1F1C4_IS2A : BOOL := false;
    C1F1C4_IS2B : BOOL := false;
    Not_Connected : BOOL := false;
  END_VAR
  VAR
    FB_C1F1C4_Part_Detection_x2 : Part Detection x2;
  END_VAR

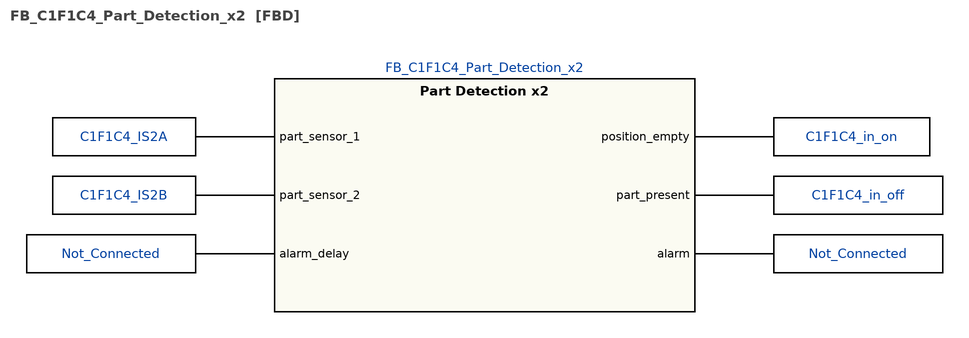
(* FBD diagram, written out as Structured Text *)
FB_C1F1C4_Part_Detection_x2(part_sensor_1 := C1F1C4_IS2A, part_sensor_2 := C1F1C4_IS2B, alarm_delay := Not_Connected);
C1F1C4_in_on := FB_C1F1C4_Part_Detection_x2.position_empty;
C1F1C4_in_off := FB_C1F1C4_Part_Detection_x2.part_present;
Not_Connected := FB_C1F1C4_Part_Detection_x2.alarm;
END_PROGRAM

PROGRAM FB_Zone_1
  VAR_EXTERNAL
    C1R1_book_zone_1 : BOOL := false;
    C1R1_unbook_zone_1 : BOOL := false;
    C1R1_zone_1_booked : BOOL := false;
    Not_Connected : BOOL := false;
  END_VAR
  VAR
    FB_Zone_1 : Zone booking x1;
  END_VAR

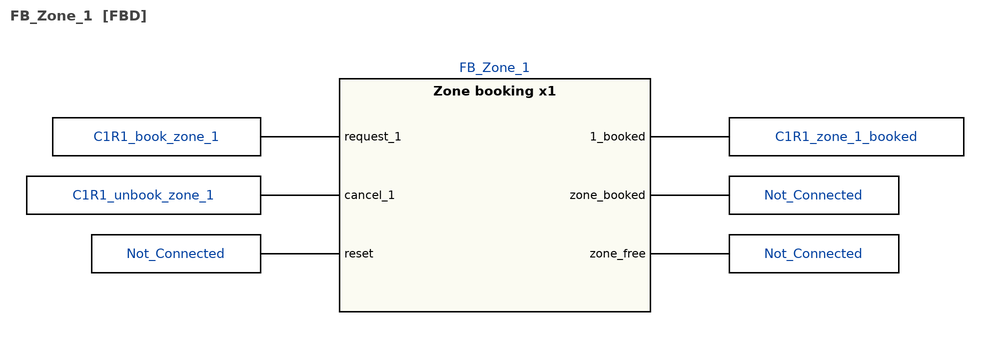
(* FBD diagram, written out as Structured Text *)
FB_Zone_1(request_1 := C1R1_book_zone_1, cancel_1 := C1R1_unbook_zone_1, reset := Not_Connected);
C1R1_zone_1_booked := FB_Zone_1.1_booked;
Not_Connected := FB_Zone_1.zone_booked;
Not_Connected := FB_Zone_1.zone_free;
END_PROGRAM

PROGRAM FB_Zone_2
  VAR_EXTERNAL
    C1R1_book_zone_2 : BOOL := false;
    C1R1_unbook_zone_2 : BOOL := false;
    C1R1_zone_2_booked : BOOL := false;
    C1F1_book_zone_2 : BOOL := false;
    C1F1_unbook_zone_2 : BOOL := false;
    C1F1_zone_2_booked : BOOL := false;
    C1C1_book_zone_2 : BOOL := false;
    C1C1_unbook_zone_2 : BOOL := false;
    C1C1_zone_2_booked : BOOL := false;
    Not_Connected : BOOL := false;
  END_VAR
  VAR
    FB_Zone_2 : Zone booking x3;
  END_VAR

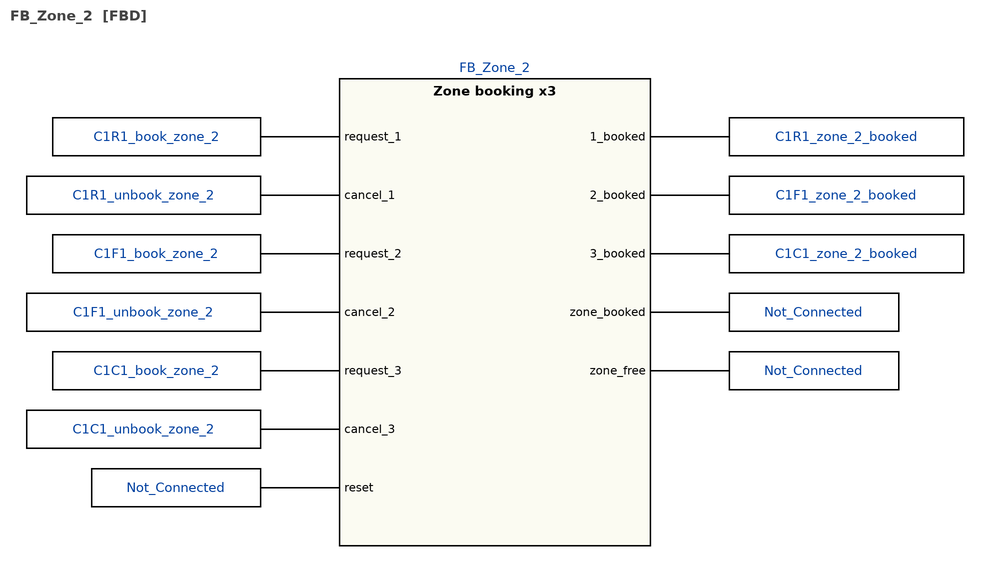
(* FBD diagram, written out as Structured Text *)
FB_Zone_2(request_1 := C1R1_book_zone_2, cancel_1 := C1R1_unbook_zone_2, request_2 := C1F1_book_zone_2, cancel_2 := C1F1_unbook_zone_2, request_3 := C1C1_book_zone_2, cancel_3 := C1C1_unbook_zone_2, reset := Not_Connected);
C1R1_zone_2_booked := FB_Zone_2.1_booked;
C1F1_zone_2_booked := FB_Zone_2.2_booked;
C1C1_zone_2_booked := FB_Zone_2.3_booked;
Not_Connected := FB_Zone_2.zone_booked;
Not_Connected := FB_Zone_2.zone_free;
END_PROGRAM

PROGRAM FB_Zone_3
  VAR_EXTERNAL
    C1R1_book_zone_3 : BOOL := false;
    C1R1_unbook_zone_3 : BOOL := false;
    C1R1_zone_3_booked : BOOL := false;
    C1F1_book_zone_3 : BOOL := false;
    C1F1_unbook_zone_3 : BOOL := false;
    C1F1_zone_3_booked : BOOL := false;
    C1C1_book_zone_3 : BOOL := false;
    C1C1_unbook_zone_3 : BOOL := false;
    C1C1_zone_3_booked : BOOL := false;
    Not_Connected : BOOL := false;
  END_VAR
  VAR
    FB_Zone_3 : Zone booking x3;
  END_VAR

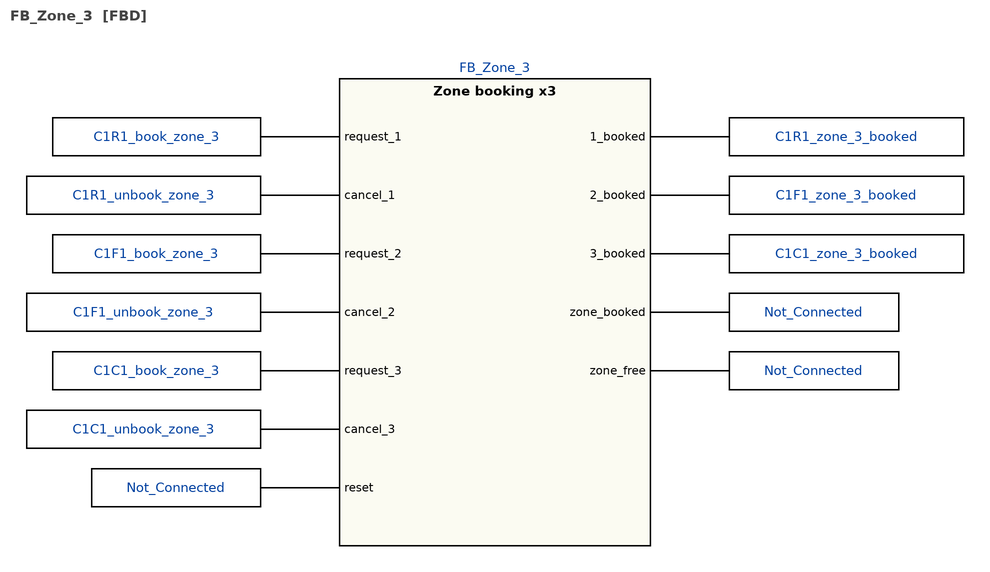
(* FBD diagram, written out as Structured Text *)
FB_Zone_3(request_1 := C1R1_book_zone_3, cancel_1 := C1R1_unbook_zone_3, request_2 := C1F1_book_zone_3, cancel_2 := C1F1_unbook_zone_3, request_3 := C1C1_book_zone_3, cancel_3 := C1C1_unbook_zone_3, reset := Not_Connected);
C1R1_zone_3_booked := FB_Zone_3.1_booked;
C1F1_zone_3_booked := FB_Zone_3.2_booked;
C1C1_zone_3_booked := FB_Zone_3.3_booked;
Not_Connected := FB_Zone_3.zone_booked;
Not_Connected := FB_Zone_3.zone_free;
END_PROGRAM

PROGRAM IL_C1_41
  VAR_EXTERNAL
    C1F1C1_in_home : BOOL := false;
    C1R1C4_in_on : BOOL := false;
    C1C1_zone_2_booked : BOOL := false;
    C1C1_zone_3_booked : BOOL := false;
    C1C1C1_IL_to_41 : BOOL := false;
  END_VAR

